INTERFACE I_InputSource

METHOD AddClient : BOOL
VAR_OUTPUT
	nClientID: LWORD;
END_VAR
END_METHOD

METHOD Call : BOOL
END_METHOD

METHOD ClientDone : BOOL
VAR_INPUT
	nClientID: LWORD;
END_VAR
END_METHOD

METHOD GetData : BOOL
VAR_INPUT
	nElement: UDINT;
	pInputs: PVOID;
	nInputsSize: UDINT;
END_VAR
VAR_OUTPUT
	nTimestamp: ULINT;
	nContext: DWORD;
END_VAR
END_METHOD

METHOD NewDataAvailable : BOOL
VAR_INPUT
	nLastDataHandle: ULINT;
END_VAR
END_METHOD

PROPERTY eDataState : E_DataSourceState
GET
END_GET
END_PROPERTY

PROPERTY bReadNewData : BOOL
GET
END_GET
END_PROPERTY

PROPERTY nDataHandle : ULINT
GET
END_GET
END_PROPERTY

PROPERTY nElements : UDINT
GET
END_GET
END_PROPERTY

END_INTERFACE

(* stored: Itf I_InputSource: Id eab3ba12-2b34-4309-8253-8d2655868ba7
   Method AddClient: Id cccb7723-70e6-4120-8b3c-8c5381caeb91
   Method Call: Id 428459df-9036-4cb8-bf66-9051db543df5
   Method ClientDone: Id 51c0ed6c-7086-4e85-af34-f26a7d767a94
   Method GetData: Id 3e1c17b3-f5dd-4194-b0ec-eb6724247956
   Method NewDataAvailable: Id 5d78ae1a-706b-4733-bff4-ab6e99a1a544
   Property eDataState: Id d5ccac1d-cfd7-4b5b-9a8d-199766c439be
   Get Get: Id 6f284543-d11e-4574-9fbc-9c307e1d0fe1
   Property bReadNewData: Id b91347d1-445c-461d-aa57-f30dca5d7c30
   Get Get: Id 18a24e86-6742-4f09-b775-a0fa85397c98
   Property nDataHandle: Id 93e8006a-65e0-43f4-9772-757b73828abb
   Get Get: Id 03494a5d-0e88-463f-9e00-d2879d761017
   Property nElements: Id 07393704-d060-481f-89b2-359a8da8708b
   Get Get: Id 8a3160b0-e3cf-4a4d-9b71-27480662686b *)
